{attribute 'qualified_only'}
{attribute 'strict'}
TYPE PLCOpenCallState :
(
	ATN_PLCOPEN_FUB_IDLE := 0,
	ATN_PLCOPEN_FUB_NEW_COMMAND,
	ATN_PLCOPEN_FUB_ABORTED,
	ATN_PLCOPEN_FUB_ABORT_OLD,
	ATN_PLCOPEN_FUB_STATUS,
	ATN_PLCOPEN_FUB_WRITE_PAR,
	ATN_PLCOPEN_FUB_SET_COMMAND,
	ATN_PLCOPEN_FUB_WORKING,
	ATN_PLCOPEN_FUB_CLEANUP,
	ATN_PLCOPEN_FUB_DONE
);
END_TYPE

(* stored: Version 1.1.0.1, ProductVersion 3.1.4024.12
   EnumerationTextList PLCOpenCallState: Id {3ae6e054-32d2-4fc8-9116-cc770a82905a} *)
